TEXTLIST Tensometr
  0 = '50t'
  1 = '100t'
   = ''
END_TEXTLIST

(* stored: Version 1.1.0.1, ProductVersion 3.1.4024.16
   TextList Tensometr: Id {356997b1-dd69-4585-aef7-fc53970ebe34} *)
